# EPICS autosave request: iocBoot/ioc13bma_linux/auto_settings.req
file "Keithley2kDMM_mf10_settings.req", P=$(P), Dmm=DMM1
file "Keithley2kDMM_mf10_settings.req", P=$(P), Dmm=DMM2
file "table_settings.req",              P=$(P), T=MON:t1, Q=MON:T1
file "mono_pid_control_settings.req",   P=$(P), PID=mono_pid1
file "auto_shutter_settings.req",       P=$(P), SHUT=FOE
file "auto_shutter_settings.req",       P=$(P), SHUT=BMC
file "auto_shutter_settings.req",       P=$(P), SHUT=BMD
file "MPC_settings.req",                P=$(P), PUMP=ip8:
file "MPC_settings.req",                P=$(P), PUMP=ip9:
file "TSP_settings.req",                P=$(P), TSP=tsp1:
file "scan_settings.req",               P=$(P), S=scan1
file "scan_settings.req",               P=$(P), S=scan2
file "scan_settings.req",               P=$(P), S=scan3
file "scan_settings.req",               P=$(P), S=scan4
file "saveData_settings.req",           P=$(P)
file "Galil_settings.req",               P=$(P)
file "Energy_settings.req",             P=$(P), EN=E
file "E1608_settings.req",              P=$(E1608_PREFIX)
file "calc_GSECARS.req",                P=$(P)
